FUNCTION_BLOCK switch_var_to_ev
  (* Standard: 61499-2 *)
  (* Version 11-01-12, GASR *)
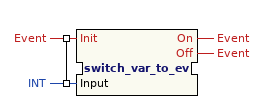
  EVENT_INPUT
    Init WITH Input;
  END_EVENT
  EVENT_OUTPUT
    On;
    Off;
  END_EVENT
  VAR_INPUT
    Input : INT;
  END_VAR
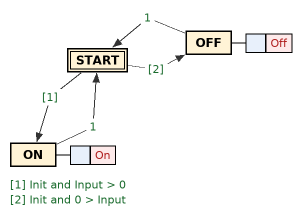
  EC_STATES
    START;
    ON : -> On;
    OFF : -> Off;
  END_STATES
  EC_TRANSITIONS
    START TO ON := Init and Input > 0;
    START TO OFF := Init and 0 > Input;
    ON TO START := 1;
    OFF TO START := 1;
  END_TRANSITIONS
END_FUNCTION_BLOCK
